RoboDK station: PenHolder.rdk

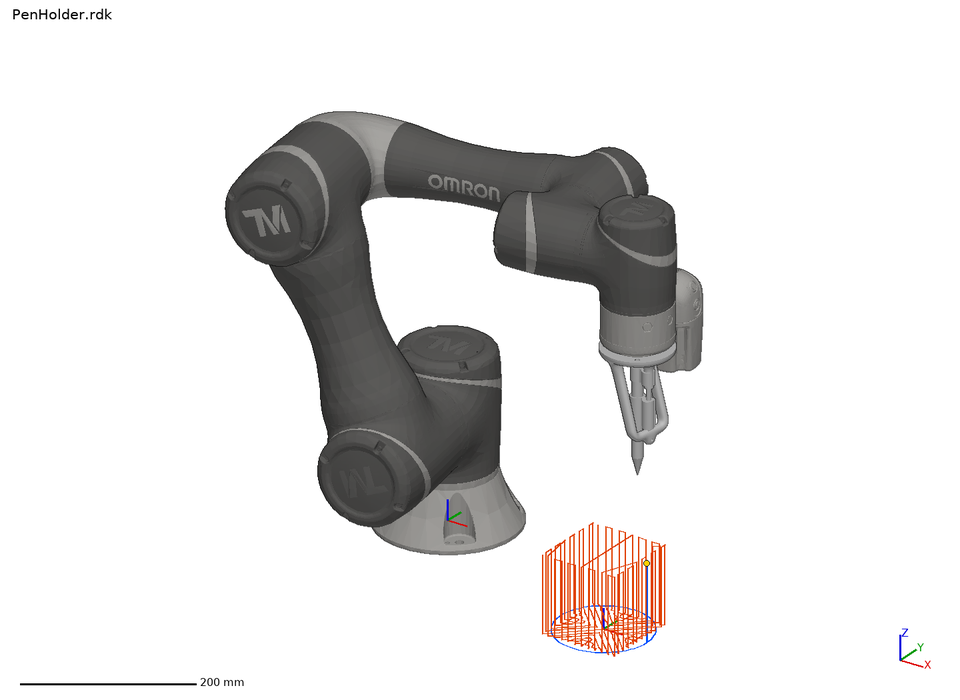
[picture v0: the station drawn from its stored meshes, robots at their saved joint values, targets as dots, program paths as lines]
Station PenHolder (saved by RoboDK 5.6.7). Poses are relative to the parent item; angles as X-Y-Z fixed-axis rotations.
  - frame Omron TM5-700 Base at (0, 0, 0) mm
    - robot Omron TM5-700: 6 axes, payload 6 kg, reach 700 mm, repeatability 0.05 mm, weight 22.1 kg
        modified DH rows (alpha deg, a mm, theta deg, d mm): 0, 0, 0, 145.2; 90, 0, 90, 0; 0, 329, 0, 0; 0, 311, -90, 122.3; -90, 0, 0, 106.5; 90, 0, 180, 114.15
        joint limits [-270, -180, -155, -180, -180, -270] to [270, 180, 155, 180, 180, 270]; home [0, 0, 90, -90, 90, 0]; saved at [8.928, -21.013, 110.905, 0.108, 90, -86.327]
      - tool PenHolderTCP, TCP at (0, 0, 163) mm, size 163 x 88.1 x 88.4 mm, geometry from PenHolderTCP.stl
  - frame Canvas at (306.28, -129, 0) mm
    - object circle at (0, 0, 0) mm, geometry from pter
    - object pattern at (0, 0, 0) mm, geometry from amag
  - machining project circle Settings: rotZ(0) | rotX(0)*rotY(0) | rotz(0) | onStart | onPathStart | onApproach | onPoint | onRetract | onFinish | SetRPM(%1) | SetTool(%1) | Extruder(%1) | default | default | OutOnMov(%1) | OutOffMov(%1) | onPathFinish | M_RunCode(%1)
  - program circle (86 instructions, listed below)
  - machining project pattern Settings: rotZ(0) | rotX(0)*rotY(0) | rotz(0) | onStart | onPathStart | onApproach | onPoint | onRetract | onFinish | SetRPM(%1) | SetTool(%1) | Extruder(%1) | default | default | OutOnMov(%1) | OutOffMov(%1) | onPathFinish | M_RunCode(%1)
  - program patternLinear (449 instructions, listed below)
  - Python program Prog3 (listed below)
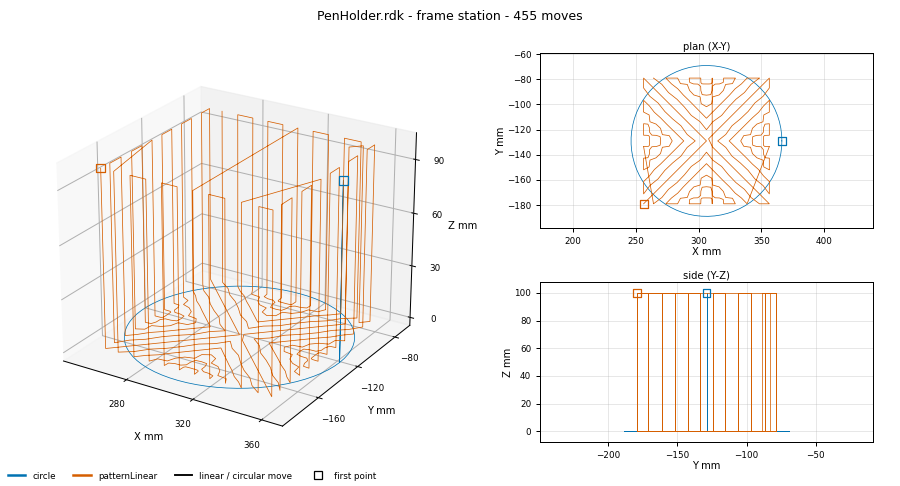
[picture p0: tool path of PenHolder.rdk in frame station, 455 of 455 moves have a stored position in this frame; points joined in program order, loops and branches not executed]

--- program circle (robot Omron TM5-700) ---
  Smooth(1)
  Set speed (1000.0 mm/s)
  Set Ref.: Canvas
  Set Tool: PenHolderTCP
  Show PenHolderTCP
  MoveJ 1 to (60, 0, 100) mm, rotated rx -180 ry 0 rz -180 deg; joints [-1.045, -5.926, 113.769, -17.843, 90, -91.045]
  MoveL 2 to (60, 0, 100) mm, rotated rx -180 ry 0 rz -180 deg; joints [-1.045, -5.926, 113.769, -17.843, 90, -91.045]
  MoveL 3 to (60, 0, 0) mm, rotated rx -180 ry 0 rz -180 deg; joints [-1.045, 3.646, 125.512, -39.158, 90, -91.045]
  MoveL 4 to (60, 0, 0) mm, rotated rx -180 ry 0 rz -180 deg; joints [-1.045, 3.646, 125.512, -39.158, 90, -91.045]
  Set speed (50.0 mm/s)
  MoveL 5 to (59.78, 5.16, 0) mm, rotated rx -180 ry 0 rz -180 deg; joints [-0.241, 3.314, 125.871, -39.185, 90, -90.241]
  MoveL 6 to (59.11, 10.28, 0) mm, rotated rx -180 ry 0 rz -180 deg; joints [0.562, 2.919, 126.295, -39.215, 90, -89.438]
  MoveL 7 to (58.01, 15.32, 0) mm, rotated rx -180 ry 0 rz -180 deg; joints [1.361, 2.462, 126.782, -39.244, 90, -88.639]
  MoveL 8 to (56.48, 20.25, 0) mm, rotated rx -180 ry 0 rz 180 deg; joints [2.153, 1.943, 127.328, -39.271, 90, -87.847]
  MoveL 9 to (54.53, 25.03, 0) mm, rotated rx -180 ry 0 rz -180 deg; joints [2.934, 1.364, 127.93, -39.294, 90, -87.066]
  MoveL 10 to (52.18, 29.63, 0) mm, rotated rx -180 ry 0 rz -180 deg; joints [3.7, 0.726, 128.584, -39.31, 90, -86.3]
  MoveL 11 to (49.44, 34, 0) mm, rotated rx -180 ry 0 rz -180 deg; joints [4.448, 0.029, 129.287, -39.316, 90, -85.552]
  MoveL 12 to (46.33, 38.13, 0) mm, rotated rx -180 ry 0 rz -180 deg; joints [5.173, -0.723, 130.033, -39.31, 90, -84.827]
  MoveL 13 to (42.88, 41.97, 0) mm, rotated rx -180 ry 0 rz -180 deg; joints [5.872, -1.529, 130.818, -39.288, 90, -84.128]
  MoveL 14 to (39.11, 45.5, 0) mm, rotated rx -180 ry 0 rz -180 deg; joints [6.54, -2.388, 131.636, -39.248, 90, -83.46]
  MoveL 15 to (35.06, 48.69, 0) mm, rotated rx -180 ry 0 rz -180 deg; joints [7.173, -3.295, 132.482, -39.187, 90, -82.827]
  MoveL 16 to (30.74, 51.53, 0) mm, rotated rx -180 ry 0 rz -180 deg; joints [7.765, -4.25, 133.351, -39.101, 90, -82.235]
  MoveL 17 to (26.2, 53.98, 0) mm, rotated rx -180 ry 0 rz -180 deg; joints [8.312, -5.247, 134.236, -38.989, 90, -81.688]
  MoveL 18 to (21.46, 56.03, 0) mm, rotated rx -180 ry 0 rz -180 deg; joints [8.809, -6.284, 135.131, -38.847, 90, -81.191]
  MoveL 19 to (16.57, 57.67, 0) mm, rotated rx -180 ry 0 rz -180 deg; joints [9.25, -7.355, 136.03, -38.675, 90, -80.75]
  MoveL 20 to (11.55, 58.88, 0) mm, rotated rx -180 ry 0 rz -180 deg; joints [9.63, -8.455, 136.925, -38.47, 90, -80.37]
  MoveL 21 to (6.44, 59.65, 0) mm, rotated rx -180 ry 0 rz -180 deg; joints [9.942, -9.577, 137.81, -38.233, 90, -80.058]
  MoveL 22 to (1.29, 59.99, 0) mm, rotated rx -180 ry 0 rz -180 deg; joints [10.182, -10.715, 138.678, -37.963, 90, -79.818]
  MoveL 23 to (-3.87, 59.88, 0) mm, rotated rx -180 ry 0 rz -180 deg; joints [10.343, -11.858, 139.522, -37.664, 90, -79.657]
  MoveL 24 to (-9, 59.32, 0) mm, rotated rx -180 ry 0 rz -180 deg; joints [10.42, -12.999, 140.335, -37.336, 90, -79.58]
  MoveL 25 to (-14.07, 58.33, 0) mm, rotated rx -180 ry 0 rz -180 deg; joints [10.408, -14.124, 141.11, -36.986, 90, -79.592]
  MoveL 26 to (-19.03, 56.9, 0) mm, rotated rx -180 ry 0 rz 180 deg; joints [10.3, -15.223, 141.841, -36.618, 90, -79.7]
  MoveL 27 to (-23.85, 55.06, 0) mm, rotated rx -180 ry 0 rz -180 deg; joints [10.094, -16.282, 142.522, -36.24, 90, -79.906]
  MoveL 28 to (-28.5, 52.8, 0) mm, rotated rx -180 ry 0 rz -180 deg; joints [9.785, -17.285, 143.146, -35.861, 90, -80.215]
  MoveL 29 to (-32.93, 50.16, 0) mm, rotated rx -180 ry 0 rz -180 deg; joints [9.371, -18.217, 143.709, -35.491, 90, -80.629]
  MoveL 30 to (-37.12, 47.14, 0) mm, rotated rx -180 ry 0 rz -180 deg; joints [8.851, -19.064, 144.204, -35.14, 90, -81.149]
  MoveL 31 to (-41.04, 43.77, 0) mm, rotated rx -180 ry 0 rz 180 deg; joints [8.226, -19.808, 144.629, -34.82, 90, -81.774]
  MoveL 32 to (-44.65, 40.08, 0) mm, rotated rx -180 ry 0 rz -180 deg; joints [7.498, -20.437, 144.979, -34.542, 90, -82.502]
  MoveL 33 to (-47.93, 36.1, 0) mm, rotated rx -180 ry 0 rz -180 deg; joints [6.674, -20.936, 145.252, -34.316, 90, -83.326]
  MoveL 34 to (-50.85, 31.84, 0) mm, rotated rx -180 ry 0 rz -180 deg; joints [5.76, -21.295, 145.446, -34.151, 90, -84.24]
  MoveL 35 to (-53.4, 27.35, 0) mm, rotated rx -180 ry 0 rz -180 deg; joints [4.765, -21.506, 145.558, -34.053, 90, -85.235]
  MoveL 36 to (-55.56, 22.66, 0) mm, rotated rx -180 ry 0 rz -180 deg; joints [3.701, -21.563, 145.588, -34.026, 90, -86.299]
  MoveL 37 to (-57.3, 17.8, 0) mm, rotated rx -180 ry 0 rz -180 deg; joints [2.582, -21.465, 145.537, -34.072, 90, -87.418]
  MoveL 38 to (-58.62, 12.81, 0) mm, rotated rx -180 ry 0 rz -180 deg; joints [1.422, -21.215, 145.403, -34.188, 90, -88.578]
  MoveL 39 to (-59.5, 7.72, 0) mm, rotated rx -180 ry 0 rz -180 deg; joints [0.238, -20.818, 145.188, -34.37, 90, -89.762]
  MoveL 40 to (-59.94, 2.58, 0) mm, rotated rx -180 ry 0 rz -180 deg; joints [-0.954, -20.284, 144.895, -34.611, 90, -90.954]
  MoveL 41 to (-59.94, -2.58, 0) mm, rotated rx -180 ry 0 rz -180 deg; joints [-2.138, -19.623, 144.524, -34.901, 90, -92.138]
  MoveL 42 to (-59.5, -7.72, 0) mm, rotated rx -180 ry 0 rz 180 deg; joints [-3.299, -18.85, 144.081, -35.23, 90, -93.299]
  MoveL 43 to (-58.62, -12.81, 0) mm, rotated rx -180 ry 0 rz -180 deg; joints [-4.421, -17.98, 143.567, -35.587, 90, -94.421]
  MoveL 44 to (-57.3, -17.8, 0) mm, rotated rx -180 ry 0 rz -180 deg; joints [-5.492, -17.027, 142.988, -35.961, 90, -95.492]
  MoveL 45 to (-55.56, -22.66, 0) mm, rotated rx -180 ry 0 rz -180 deg; joints [-6.501, -16.008, 142.348, -36.34, 90, -96.501]
  MoveL 46 to (-53.4, -27.35, 0) mm, rotated rx -180 ry 0 rz -180 deg; joints [-7.439, -14.938, 141.654, -36.716, 90, -97.439]
  MoveL 47 to (-50.85, -31.84, 0) mm, rotated rx -180 ry 0 rz -180 deg; joints [-8.297, -13.83, 140.911, -37.08, 90, -98.297]
  MoveL 48 to (-47.93, -36.1, 0) mm, rotated rx -180 ry 0 rz 180 deg; joints [-9.071, -12.7, 140.125, -37.425, 90, -99.071]
  MoveL 49 to (-44.65, -40.08, 0) mm, rotated rx -180 ry 0 rz 180 deg; joints [-9.757, -11.557, 139.303, -37.745, 90, -99.757]
  MoveL 50 to (-41.04, -43.77, 0) mm, rotated rx -180 ry 0 rz -180 deg; joints [-10.352, -10.414, 138.452, -38.037, 90, -100.352]
  MoveL 51 to (-37.12, -47.14, 0) mm, rotated rx -180 ry 0 rz -180 deg; joints [-10.855, -9.28, 137.579, -38.298, 90, -100.855]
  MoveL 52 to (-32.93, -50.16, 0) mm, rotated rx -180 ry 0 rz -180 deg; joints [-11.266, -8.163, 136.69, -38.527, 90, -101.266]
  MoveL 53 to (-28.5, -52.8, 0) mm, rotated rx -180 ry 0 rz -180 deg; joints [-11.587, -7.07, 135.793, -38.723, 90, -101.587]
  MoveL 54 to (-23.85, -55.06, 0) mm, rotated rx -180 ry 0 rz 180 deg; joints [-11.82, -6.008, 134.895, -38.887, 90, -101.82]
  MoveL 55 to (-19.03, -56.9, 0) mm, rotated rx -180 ry 0 rz -180 deg; joints [-11.967, -4.981, 134.002, -39.021, 90, -101.967]
  MoveL 56 to (-14.07, -58.33, 0) mm, rotated rx -180 ry 0 rz -180 deg; joints [-12.032, -3.995, 133.121, -39.126, 90, -102.032]
  MoveL 57 to (-9, -59.32, 0) mm, rotated rx -180 ry 0 rz 180 deg; joints [-12.017, -3.052, 132.257, -39.205, 90, -102.017]
  MoveL 58 to (-3.87, -59.88, 0) mm, rotated rx -180 ry 0 rz -180 deg; joints [-11.927, -2.157, 131.418, -39.261, 90, -101.927]
  MoveL 59 to (1.29, -59.99, 0) mm, rotated rx -180 ry 0 rz 180 deg; joints [-11.766, -1.312, 130.608, -39.296, 90, -101.766]
  MoveL 60 to (6.44, -59.65, 0) mm, rotated rx -180 ry 0 rz 180 deg; joints [-11.537, -0.52, 129.833, -39.313, 90, -101.537]
  MoveL 61 to (11.55, -58.88, 0) mm, rotated rx -180 ry 0 rz -180 deg; joints [-11.244, 0.218, 129.098, -39.316, 90, -101.244]
  MoveL 62 to (16.57, -57.67, 0) mm, rotated rx -180 ry 0 rz -180 deg; joints [-10.892, 0.899, 128.408, -39.307, 90, -100.892]
  MoveL 63 to (21.46, -56.03, 0) mm, rotated rx -180 ry 0 rz -180 deg; joints [-10.485, 1.522, 127.767, -39.289, 90, -100.485]
  MoveL 64 to (26.2, -53.98, 0) mm, rotated rx -180 ry 0 rz -180 deg; joints [-10.026, 2.085, 127.179, -39.264, 90, -100.026]
  MoveL 65 to (30.74, -51.53, 0) mm, rotated rx -180 ry 0 rz -180 deg; joints [-9.52, 2.588, 126.648, -39.236, 90, -99.52]
  MoveL 66 to (35.06, -48.69, 0) mm, rotated rx -180 ry 0 rz -180 deg; joints [-8.97, 3.029, 126.178, -39.207, 90, -98.97]
  MoveL 67 to (39.11, -45.5, 0) mm, rotated rx -180 ry 0 rz 180 deg; joints [-8.38, 3.407, 125.77, -39.178, 90, -98.38]
  MoveL 68 to (42.88, -41.97, 0) mm, rotated rx -180 ry 0 rz -180 deg; joints [-7.753, 3.722, 125.429, -39.151, 90, -97.753]
  MoveL 69 to (46.33, -38.13, 0) mm, rotated rx -180 ry 0 rz -180 deg; joints [-7.094, 3.973, 125.155, -39.128, 90, -97.094]
  MoveL 70 to (49.44, -34, 0) mm, rotated rx -180 ry 0 rz -180 deg; joints [-6.406, 4.16, 124.95, -39.11, 90, -96.406]
  MoveL 71 to (52.18, -29.63, 0) mm, rotated rx -180 ry 0 rz 180 deg; joints [-5.691, 4.282, 124.816, -39.098, 90, -95.691]
  MoveL 72 to (54.53, -25.03, 0) mm, rotated rx -180 ry 0 rz -180 deg; joints [-4.954, 4.338, 124.754, -39.092, 90, -94.954]
  MoveL 73 to (56.48, -20.25, 0) mm, rotated rx -180 ry 0 rz -180 deg; joints [-4.197, 4.33, 124.764, -39.093, 90, -94.197]
  MoveL 74 to (58.01, -15.32, 0) mm, rotated rx -180 ry 0 rz 180 deg; joints [-3.425, 4.256, 124.845, -39.101, 90, -93.425]
  MoveL 75 to (59.11, -10.28, 0) mm, rotated rx -180 ry 0 rz -180 deg; joints [-2.64, 4.117, 124.997, -39.114, 90, -92.64]
  MoveL 76 to (59.78, -5.16, 0) mm, rotated rx -180 ry 0 rz -180 deg; joints [-1.846, 3.914, 125.22, -39.134, 90, -91.846]
  MoveL 77 to (60, 0, 0) mm, rotated rx -180 ry 0 rz -180 deg; joints [-1.045, 3.646, 125.512, -39.158, 90, -91.045]
  Set speed (1000.0 mm/s)
  MoveL 78 to (60, 0, 0) mm, rotated rx -180 ry 0 rz -180 deg; joints [-1.045, 3.646, 125.512, -39.158, 90, -91.045]
  MoveL 79 to (60, 0, 100) mm, rotated rx -180 ry 0 rz -180 deg; joints [-1.045, -5.926, 113.769, -17.843, 90, -91.045]

--- program patternLinear (robot Omron TM5-700) ---
  Smooth(1)
  Set speed (1000.0 mm/s)
  Set Ref.: Canvas
  Set Tool: PenHolderTCP
  Show PenHolderTCP
  MoveJ 1 to (-50, -50, 100) mm, rotated rx -180 ry 0 rz -180 deg; joints [-11.902, -21.555, 125.328, -13.773, 90, -101.902]
  MoveL 2 to (-50, -50, 100) mm, rotated rx -180 ry 0 rz -180 deg; joints [-11.902, -21.555, 125.328, -13.773, 90, -101.902]
  MoveL 3 to (-50, -50, 0) mm, rotated rx -180 ry 0 rz -180 deg; joints [-11.902, -11.308, 139.12, -37.811, 90, -101.902]
  MoveL 4 to (-50, -50, 0) mm, rotated rx -180 ry 0 rz -180 deg; joints [-11.902, -11.308, 139.12, -37.811, 90, -101.902]
  Set speed (50.0 mm/s)
  MoveL 5 to (-7.14, -7.14, 0) mm, rotated rx -180 ry 0 rz -180 deg; joints [-2.625, -7.772, 136.372, -38.6, 90, -92.625]
  MoveL 6 to (0, 0, 0) mm, rotated rx -180 ry 0 rz -180 deg; joints [-1.248, -6.997, 135.732, -38.735, 90, -91.248]
  MoveL 7 to (-50, 50, 0) mm, rotated rx -180 ry 0 rz -180 deg; joints [9.999, -22.769, 146.216, -33.447, 90, -80.001]
  Set speed (1000.0 mm/s)
  MoveL 8 to (-50, 50, 0) mm, rotated rx -180 ry 0 rz -180 deg; joints [9.999, -22.769, 146.216, -33.447, 90, -80.001]
  MoveL 9 to (-50, 50, 100) mm, rotated rx -180 ry 0 rz -180 deg; joints [9.999, -32.206, 130.792, -8.586, 90, -80.001]
  Set speed (1000.0 mm/s)
  MoveL 10 to (-50, 42.13, 100) mm, rotated rx -180 ry 0 rz 180 deg; joints [8.143, -31.588, 130.523, -8.935, 90, -81.857]
  MoveL 11 to (-50, 42.13, 0) mm, rotated rx -180 ry 0 rz 180 deg; joints [8.143, -22.062, 145.851, -33.789, 90, -81.857]
  MoveL 12 to (-50, 42.13, 0) mm, rotated rx -180 ry 0 rz 180 deg; joints [8.143, -22.062, 145.851, -33.789, 90, -81.857]
  Set speed (50.0 mm/s)
  MoveL 13 to (-45.03, 35.49, 0) mm, rotated rx -180 ry 0 rz -180 deg; joints [6.459, -20.118, 144.802, -34.684, 90, -83.541]
  MoveL 14 to (-38.5, 30.21, 0) mm, rotated rx -180 ry 0 rz 180 deg; joints [5.121, -17.972, 143.562, -35.59, 90, -84.879]
  MoveL 15 to (-33.12, 23.42, 0) mm, rotated rx -180 ry 0 rz -180 deg; joints [3.551, -16.051, 142.375, -36.325, 90, -86.449]
  MoveL 16 to (-26.96, 17.54, 0) mm, rotated rx -180 ry 0 rz -180 deg; joints [2.241, -14.099, 141.093, -36.994, 90, -87.759]
  MoveL 17 to (-20.31, 12.08, 0) mm, rotated rx -180 ry 0 rz -180 deg; joints [1.081, -12.149, 139.732, -37.583, 90, -88.919]
  MoveL 18 to (-15.34, 5.14, 0) mm, rotated rx -180 ry 0 rz -180 deg; joints [-0.307, -10.493, 138.511, -38.018, 90, -90.307]
  MoveL 19 to (-8.95, 0, 0) mm, rotated rx -180 ry 0 rz -180 deg; joints [-1.285, -8.749, 137.159, -38.411, 90, -91.285]
  MoveL 20 to (-15.34, -5.14, 0) mm, rotated rx -180 ry 0 rz 180 deg; joints [-2.311, -9.566, 137.801, -38.235, 90, -92.311]
  MoveL 21 to (-20.31, -12.08, 0) mm, rotated rx -180 ry 0 rz -180 deg; joints [-3.706, -9.896, 138.056, -38.16, 90, -93.706]
  MoveL 22 to (-26.96, -17.54, 0) mm, rotated rx -180 ry 0 rz 180 deg; joints [-4.869, -10.668, 138.643, -37.975, 90, -94.869]
  MoveL 23 to (-33.12, -23.42, 0) mm, rotated rx -180 ry 0 rz -180 deg; joints [-6.145, -11.262, 139.085, -37.824, 90, -96.145]
  MoveL 24 to (-38.5, -30.21, 0) mm, rotated rx -180 ry 0 rz -180 deg; joints [-7.619, -11.553, 139.3, -37.746, 90, -97.619]
  MoveL 25 to (-45.03, -35.49, 0) mm, rotated rx -180 ry 0 rz -180 deg; joints [-8.859, -12.203, 139.771, -37.568, 90, -98.859]
  MoveL 26 to (-50, -42.13, 0) mm, rotated rx -180 ry 0 rz 180 deg; joints [-10.35, -12.334, 139.864, -37.531, 90, -100.35]
  Set speed (1000.0 mm/s)
  MoveL 27 to (-50, -42.13, 0) mm, rotated rx -180 ry 0 rz 180 deg; joints [-10.35, -12.334, 139.864, -37.531, 90, -100.35]
  MoveL 28 to (-50, -42.13, 100) mm, rotated rx -180 ry 0 rz 180 deg; joints [-10.35, -22.561, 125.923, -13.362, 90, -100.35]
  Set speed (1000.0 mm/s)
  MoveL 29 to (-50, -32.32, 100) mm, rotated rx -180 ry 0 rz -180 deg; joints [-8.369, -23.786, 126.624, -12.838, 90, -98.369]
  MoveL 30 to (-50, -32.32, 0) mm, rotated rx -180 ry 0 rz -180 deg; joints [-8.369, -13.596, 140.75, -37.154, 90, -98.369]
  MoveL 31 to (-50, -32.32, 0) mm, rotated rx -180 ry 0 rz -180 deg; joints [-8.369, -13.596, 140.75, -37.154, 90, -98.369]
  Set speed (50.0 mm/s)
  MoveL 32 to (-45.4, -27.84, 0) mm, rotated rx -180 ry 0 rz -180 deg; joints [-7.325, -13.221, 140.49, -37.269, 90, -97.325]
  MoveL 33 to (-41.5, -22.82, 0) mm, rotated rx -180 ry 0 rz -180 deg; joints [-6.208, -13.025, 140.354, -37.328, 90, -96.208]
  MoveL 34 to (-36.52, -18.38, 0) mm, rotated rx -180 ry 0 rz -180 deg; joints [-5.205, -12.513, 139.992, -37.479, 90, -95.205]
  MoveL 35 to (-22.58, -4.47, 0) mm, rotated rx -180 ry 0 rz -180 deg; joints [-2.237, -11.097, 138.963, -37.866, 90, -92.237]
  MoveL 36 to (-18.05, 0, 0) mm, rotated rx -180 ry 0 rz -180 deg; joints [-1.325, -10.589, 138.583, -37.995, 90, -91.325]
  MoveL 37 to (-31.87, 13.57, 0) mm, rotated rx -180 ry 0 rz -180 deg; joints [1.442, -14.841, 141.59, -36.749, 90, -88.558]
  MoveL 38 to (-36.52, 18.38, 0) mm, rotated rx -180 ry 0 rz 180 deg; joints [2.504, -16.38, 142.584, -36.204, 90, -87.496]
  MoveL 39 to (-41.5, 22.82, 0) mm, rotated rx -180 ry 0 rz -180 deg; joints [3.534, -18.009, 143.585, -35.575, 90, -86.466]
  MoveL 40 to (-45.4, 27.84, 0) mm, rotated rx -180 ry 0 rz -180 deg; joints [4.724, -19.478, 144.442, -34.964, 90, -85.276]
  MoveL 41 to (-50, 32.32, 0) mm, rotated rx -180 ry 0 rz -180 deg; joints [5.85, -21.117, 145.35, -34.233, 90, -84.15]
  Set speed (1000.0 mm/s)
  MoveL 42 to (-50, 32.32, 0) mm, rotated rx -180 ry 0 rz -180 deg; joints [5.85, -21.117, 145.35, -34.233, 90, -84.15]
  MoveL 43 to (-50, 32.32, 100) mm, rotated rx -180 ry 0 rz -180 deg; joints [5.85, -30.754, 130.152, -9.398, 90, -84.15]
  Set speed (1000.0 mm/s)
  MoveL 44 to (-50, 22.96, 100) mm, rotated rx -180 ry 0 rz -180 deg; joints [3.687, -29.894, 129.758, -9.864, 90, -86.313]
  MoveL 45 to (-50, 22.96, 0) mm, rotated rx -180 ry 0 rz -180 deg; joints [3.687, -20.153, 144.822, -34.669, 90, -86.313]
  MoveL 46 to (-50, 22.96, 0) mm, rotated rx -180 ry 0 rz -180 deg; joints [3.687, -20.153, 144.822, -34.669, 90, -86.313]
  Set speed (50.0 mm/s)
  MoveL 47 to (-45.6, 20.68, 0) mm, rotated rx -180 ry 0 rz -180 deg; joints [3.11, -18.807, 144.055, -35.248, 90, -86.89]
  MoveL 48 to (-44.95, 15.25, 0) mm, rotated rx -180 ry 0 rz -180 deg; joints [1.888, -18.079, 143.626, -35.547, 90, -88.112]
  MoveL 49 to (-40.17, 13.45, 0) mm, rotated rx -180 ry 0 rz -180 deg; joints [1.46, -16.749, 142.815, -36.066, 90, -88.54]
  MoveL 50 to (-36.57, 10.06, 0) mm, rotated rx -180 ry 0 rz -180 deg; joints [0.716, -15.57, 142.067, -36.497, 90, -89.284]
  MoveL 51 to (-35.06, 5.02, 0) mm, rotated rx -180 ry 0 rz -180 deg; joints [-0.354, -14.717, 141.508, -36.791, 90, -90.354]
  MoveL 52 to (-29.65, 4.22, 0) mm, rotated rx -180 ry 0 rz -180 deg; joints [-0.513, -13.442, 140.644, -37.202, 90, -90.513]
  MoveL 53 to (-27.24, 0, 0) mm, rotated rx -180 ry 0 rz -180 deg; joints [-1.368, -12.507, 139.988, -37.481, 90, -91.368]
  MoveL 54 to (-29.65, -4.22, 0) mm, rotated rx -180 ry 0 rz 180 deg; joints [-2.242, -12.597, 140.052, -37.455, 90, -92.242]
  MoveL 55 to (-35.06, -5.02, 0) mm, rotated rx -180 ry 0 rz -180 deg; joints [-2.452, -13.668, 140.799, -37.131, 90, -92.452]
  MoveL 56 to (-36.57, -10.06, 0) mm, rotated rx -180 ry 0 rz -180 deg; joints [-3.508, -13.447, 140.647, -37.2, 90, -93.508]
  MoveL 57 to (-40.17, -13.45, 0) mm, rotated rx -180 ry 0 rz -180 deg; joints [-4.257, -13.833, 140.913, -37.079, 90, -94.257]
  MoveL 58 to (-44.95, -15.25, 0) mm, rotated rx -180 ry 0 rz -180 deg; joints [-4.71, -14.645, 141.46, -36.815, 90, -94.71]
  MoveL 59 to (-45.6, -20.68, 0) mm, rotated rx -180 ry 0 rz -180 deg; joints [-5.858, -14.134, 141.117, -36.983, 90, -95.858]
  MoveL 60 to (-50, -22.96, 0) mm, rotated rx -180 ry 0 rz -180 deg; joints [-6.431, -14.781, 141.55, -36.769, 90, -96.431]
  Set speed (1000.0 mm/s)
  MoveL 61 to (-50, -22.96, 0) mm, rotated rx -180 ry 0 rz -180 deg; joints [-6.431, -14.781, 141.55, -36.769, 90, -96.431]
  MoveL 62 to (-50, -22.96, 100) mm, rotated rx -180 ry 0 rz -180 deg; joints [-6.431, -24.922, 127.253, -12.33, 90, -96.431]
  Set speed (1000.0 mm/s)
  MoveL 63 to (-50, -13.71, 100) mm, rotated rx -180 ry 0 rz -180 deg; joints [-4.47, -26.01, 127.835, -11.824, 90, -94.47]
  MoveL 64 to (-50, -13.71, 0) mm, rotated rx -180 ry 0 rz -180 deg; joints [-4.47, -15.93, 142.299, -36.368, 90, -94.47]
  MoveL 65 to (-50, -13.71, 0) mm, rotated rx -180 ry 0 rz -180 deg; joints [-4.47, -15.93, 142.299, -36.368, 90, -94.47]
  Set speed (50.0 mm/s)
  MoveL 66 to (-46.56, -13.35, 0) mm, rotated rx -180 ry 0 rz -180 deg; joints [-4.337, -15.221, 141.84, -36.619, 90, -94.337]
  MoveL 67 to (-45.35, -10.35, 0) mm, rotated rx -180 ry 0 rz -180 deg; joints [-3.684, -15.311, 141.899, -36.588, 90, -93.684]
  MoveL 68 to (-45.22, -6.89, 0) mm, rotated rx -180 ry 0 rz -180 deg; joints [-2.945, -15.685, 142.141, -36.456, 90, -92.945]
  MoveL 69 to (-43.44, -4.62, 0) mm, rotated rx -180 ry 0 rz -180 deg; joints [-2.442, -15.549, 142.053, -36.505, 90, -92.442]
  MoveL 70 to (-39.98, -4.45, 0) mm, rotated rx -180 ry 0 rz -180 deg; joints [-2.375, -14.801, 141.563, -36.763, 90, -92.375]
  MoveL 71 to (-36.83, -3.42, 0) mm, rotated rx -180 ry 0 rz -180 deg; joints [-2.133, -14.223, 141.177, -36.954, 90, -92.133]
  MoveL 72 to (-36.42, 0, 0) mm, rotated rx -180 ry 0 rz -180 deg; joints [-1.415, -14.497, 141.361, -36.864, 90, -91.415]
  MoveL 73 to (-36.83, 3.42, 0) mm, rotated rx -180 ry 0 rz -180 deg; joints [-0.696, -14.946, 141.66, -36.713, 90, -90.696]
  MoveL 74 to (-39.98, 4.45, 0) mm, rotated rx -180 ry 0 rz 180 deg; joints [-0.484, -15.765, 142.193, -36.428, 90, -90.484]
  MoveL 75 to (-43.44, 4.62, 0) mm, rotated rx -180 ry 0 rz -180 deg; joints [-0.453, -16.578, 142.709, -36.13, 90, -90.453]
  MoveL 76 to (-45.22, 6.89, 0) mm, rotated rx -180 ry 0 rz -180 deg; joints [0.042, -17.243, 143.121, -35.878, 90, -89.958]
  MoveL 77 to (-45.35, 10.35, 0) mm, rotated rx -180 ry 0 rz -180 deg; joints [0.805, -17.653, 143.37, -35.717, 90, -89.195]
  MoveL 78 to (-46.56, 13.35, 0) mm, rotated rx -180 ry 0 rz -180 deg; joints [1.474, -18.267, 143.738, -35.471, 90, -88.526]
  MoveL 79 to (-50, 13.71, 0) mm, rotated rx -180 ry 0 rz 180 deg; joints [1.576, -19.149, 144.253, -35.105, 90, -88.424]
  Set speed (1000.0 mm/s)
  MoveL 80 to (-50, 13.71, 0) mm, rotated rx -180 ry 0 rz 180 deg; joints [1.576, -19.149, 144.253, -35.105, 90, -88.424]
  MoveL 81 to (-50, 13.71, 100) mm, rotated rx -180 ry 0 rz 180 deg; joints [1.576, -28.986, 129.329, -10.343, 90, -88.424]
  Set speed (1000.0 mm/s)
  MoveL 82 to (-50, 4.55, 100) mm, rotated rx -180 ry 0 rz -180 deg; joints [-0.48, -28.037, 128.868, -10.831, 90, -90.48]
  MoveL 83 to (-50, 4.55, 0) mm, rotated rx -180 ry 0 rz -180 deg; joints [-0.48, -18.11, 143.645, -35.535, 90, -90.48]
  MoveL 84 to (-50, 4.55, 0) mm, rotated rx -180 ry 0 rz -180 deg; joints [-0.48, -18.11, 143.645, -35.535, 90, -90.48]
  Set speed (50.0 mm/s)
  MoveL 85 to (-48.78, 4.53, 0) mm, rotated rx -180 ry 0 rz -180 deg; joints [-0.482, -17.816, 143.469, -35.652, 90, -90.482]
  MoveL 86 to (-47.55, 4.49, 0) mm, rotated rx -180 ry 0 rz -180 deg; joints [-0.488, -17.523, 143.292, -35.768, 90, -90.488]
  MoveL 87 to (-46.33, 4.39, 0) mm, rotated rx -180 ry 0 rz -180 deg; joints [-0.508, -17.225, 143.11, -35.885, 90, -90.508]
  MoveL 88 to (-45.46, 3.67, 0) mm, rotated rx -180 ry 0 rz -180 deg; joints [-0.665, -16.942, 142.935, -35.993, 90, -90.665]
  MoveL 89 to (-45.34, 2.45, 0) mm, rotated rx -180 ry 0 rz -180 deg; joints [-0.93, -16.777, 142.833, -36.056, 90, -90.93]
  MoveL 90 to (-45.3, -1.23, 0) mm, rotated rx -180 ry 0 rz 180 deg; joints [-1.727, -16.354, 142.568, -36.214, 90, -91.727]
  MoveL 91 to (-45.34, -2.45, 0) mm, rotated rx -180 ry 0 rz -180 deg; joints [-1.992, -16.222, 142.484, -36.262, 90, -91.992]
  MoveL 92 to (-45.46, -3.67, 0) mm, rotated rx -180 ry 0 rz -180 deg; joints [-2.256, -16.111, 142.414, -36.303, 90, -92.256]
  MoveL 93 to (-46.33, -4.39, 0) mm, rotated rx -180 ry 0 rz -180 deg; joints [-2.419, -16.223, 142.485, -36.262, 90, -92.419]
  MoveL 94 to (-47.55, -4.49, 0) mm, rotated rx -180 ry 0 rz -180 deg; joints [-2.452, -16.488, 142.652, -36.164, 90, -92.452]
  MoveL 95 to (-50, -4.55, 0) mm, rotated rx -180 ry 0 rz -180 deg; joints [-2.488, -17.04, 142.996, -35.956, 90, -92.488]
  Set speed (1000.0 mm/s)
  MoveL 96 to (-50, -4.55, 0) mm, rotated rx -180 ry 0 rz -180 deg; joints [-2.488, -17.04, 142.996, -35.956, 90, -92.488]
  MoveL 97 to (-50, -4.55, 100) mm, rotated rx -180 ry 0 rz -180 deg; joints [-2.488, -27.048, 128.372, -11.324, 90, -92.488]
  Set speed (1000.0 mm/s)
  MoveL 98 to (-42.13, -50, 100) mm, rotated rx -180 ry 0 rz -180 deg; joints [-11.586, -20.105, 124.44, -14.335, 90, -101.586]
  MoveL 99 to (-42.13, -50, 0) mm, rotated rx -180 ry 0 rz 180 deg; joints [-11.586, -9.849, 138.02, -38.171, 90, -101.586]
  MoveL 100 to (-42.13, -50, 0) mm, rotated rx -180 ry 0 rz 180 deg; joints [-11.586, -9.849, 138.02, -38.171, 90, -101.586]
  Set speed (50.0 mm/s)
  MoveL 101 to (-35.49, -45.03, 0) mm, rotated rx -180 ry 0 rz -180 deg; joints [-10.398, -9.233, 137.541, -38.309, 90, -100.398]
  MoveL 102 to (-30.21, -38.5, 0) mm, rotated rx -180 ry 0 rz -180 deg; joints [-8.991, -9.009, 137.365, -38.356, 90, -98.991]
  MoveL 103 to (-23.42, -33.12, 0) mm, rotated rx -180 ry 0 rz -180 deg; joints [-7.787, -8.335, 136.829, -38.494, 90, -97.787]
  MoveL 104 to (-17.54, -26.96, 0) mm, rotated rx -180 ry 0 rz -180 deg; joints [-6.495, -7.877, 136.458, -38.581, 90, -96.495]
  MoveL 105 to (-12.08, -20.31, 0) mm, rotated rx -180 ry 0 rz -180 deg; joints [-5.149, -7.505, 136.153, -38.648, 90, -95.149]
  MoveL 106 to (-5.14, -15.34, 0) mm, rotated rx -180 ry 0 rz -180 deg; joints [-4.127, -6.661, 135.45, -38.789, 90, -94.127]
  MoveL 107 to (0, -8.95, 0) mm, rotated rx -180 ry 0 rz 180 deg; joints [-2.896, -6.254, 135.106, -38.852, 90, -92.896]
  MoveL 108 to (5.14, -15.34, 0) mm, rotated rx -180 ry 0 rz -180 deg; joints [-3.995, -4.762, 133.809, -39.046, 90, -93.995]
  MoveL 109 to (12.08, -20.31, 0) mm, rotated rx -180 ry 0 rz -180 deg; joints [-4.773, -3.106, 132.307, -39.201, 90, -94.773]
  MoveL 110 to (17.54, -26.96, 0) mm, rotated rx -180 ry 0 rz -180 deg; joints [-5.823, -1.61, 130.895, -39.285, 90, -95.823]
  MoveL 111 to (23.42, -33.12, 0) mm, rotated rx -180 ry 0 rz -180 deg; joints [-6.741, -0.115, 129.431, -39.316, 90, -96.741]
  MoveL 112 to (30.21, -38.5, 0) mm, rotated rx -180 ry 0 rz 180 deg; joints [-7.476, 1.433, 127.858, -39.292, 90, -97.476]
  MoveL 113 to (35.49, -45.03, 0) mm, rotated rx -180 ry 0 rz -180 deg; joints [-8.39, 2.802, 126.421, -39.223, 90, -98.39]
  MoveL 114 to (42.13, -50, 0) mm, rotated rx -180 ry 0 rz -180 deg; joints [-8.999, 4.232, 124.871, -39.103, 90, -98.999]
  Set speed (1000.0 mm/s)
  MoveL 115 to (42.13, -50, 0) mm, rotated rx -180 ry 0 rz -180 deg; joints [-8.999, 4.232, 124.871, -39.103, 90, -98.999]
  MoveL 116 to (42.13, -50, 100) mm, rotated rx -180 ry 0 rz -180 deg; joints [-8.999, -5.286, 113.198, -17.912, 90, -98.999]
  Set speed (1000.0 mm/s)
  MoveL 117 to (50, -50, 100) mm, rotated rx -180 ry 0 rz -180 deg; joints [-8.813, -3.961, 111.992, -18.031, 90, -98.813]
  MoveL 118 to (50, -50, 0) mm, rotated rx -180 ry 0 rz -180 deg; joints [-8.813, 5.439, 123.525, -38.964, 90, -98.813]
  MoveL 119 to (50, -50, 0) mm, rotated rx -180 ry 0 rz -180 deg; joints [-8.813, 5.439, 123.525, -38.964, 90, -98.813]
  Set speed (50.0 mm/s)
  MoveL 120 to (4.79, -4.79, 0) mm, rotated rx -180 ry 0 rz 180 deg; joints [-2.101, -5.698, 134.628, -38.93, 90, -92.101]
  MoveL 121 to (1.67, 1.67, 0) mm, rotated rx -180 ry 0 rz -180 deg; joints [-0.934, -6.809, 135.575, -38.766, 90, -90.934]
  MoveL 122 to (8.12, 8.12, 0) mm, rotated rx -180 ry 0 rz -180 deg; joints [0.26, -6.063, 134.942, -38.879, 90, -89.74]
  MoveL 123 to (40.42, 40.42, 0) mm, rotated rx -180 ry 0 rz -180 deg; joints [5.652, -1.911, 131.184, -39.273, 90, -84.348]
  Set speed (1000.0 mm/s)
  MoveL 124 to (40.42, 40.42, 0) mm, rotated rx -180 ry 0 rz -180 deg; joints [5.652, -1.911, 131.184, -39.273, 90, -84.348]
  MoveL 125 to (40.42, 40.42, 100) mm, rotated rx -180 ry 0 rz -180 deg; joints [5.652, -11.913, 118.728, -16.814, 90, -84.348]
  Set speed (1000.0 mm/s)
  MoveL 126 to (45.76, 45.76, 100) mm, rotated rx -180 ry 0 rz -180 deg; joints [6.456, -11.126, 118.114, -16.988, 90, -83.544]
  MoveL 127 to (45.76, 45.76, 0) mm, rotated rx -180 ry 0 rz -180 deg; joints [6.456, -1.17, 130.47, -39.3, 90, -83.544]
  MoveL 128 to (45.76, 45.76, 0) mm, rotated rx -180 ry 0 rz -180 deg; joints [6.456, -1.17, 130.47, -39.3, 90, -83.544]
  Set speed (50.0 mm/s)
  MoveL 129 to (50, 50, 0) mm, rotated rx -180 ry 0 rz -180 deg; joints [7.078, -0.573, 129.885, -39.312, 90, -82.922]
  Set speed (1000.0 mm/s)
  MoveL 130 to (50, 50, 0) mm, rotated rx -180 ry 0 rz -180 deg; joints [7.078, -0.573, 129.885, -39.312, 90, -82.922]
  MoveL 131 to (50, 50, 100) mm, rotated rx -180 ry 0 rz -180 deg; joints [7.078, -10.488, 117.609, -17.121, 90, -82.922]
  Set speed (1000.0 mm/s)
  MoveL 132 to (50, 42.13, 100) mm, rotated rx -180 ry 0 rz -180 deg; joints [5.778, -10.133, 117.324, -17.191, 90, -84.222]
  MoveL 133 to (50, 42.13, 0) mm, rotated rx -180 ry 0 rz -180 deg; joints [5.778, -0.241, 129.557, -39.316, 90, -84.222]
  MoveL 134 to (50, 42.13, 0) mm, rotated rx -180 ry 0 rz -180 deg; joints [5.778, -0.241, 129.557, -39.316, 90, -84.222]
  Set speed (50.0 mm/s)
  MoveL 135 to (45.03, 35.49, 0) mm, rotated rx -180 ry 0 rz -180 deg; joints [4.754, -0.833, 130.141, -39.308, 90, -85.246]
  MoveL 136 to (38.5, 30.21, 0) mm, rotated rx -180 ry 0 rz -180 deg; joints [3.949, -1.755, 131.034, -39.28, 90, -86.051]
  MoveL 137 to (33.12, 23.42, 0) mm, rotated rx -180 ry 0 rz -180 deg; joints [2.845, -2.369, 131.618, -39.249, 90, -87.155]
  MoveL 138 to (26.96, 17.54, 0) mm, rotated rx -180 ry 0 rz -180 deg; joints [1.874, -3.153, 132.351, -39.198, 90, -88.126]
  MoveL 139 to (20.31, 12.08, 0) mm, rotated rx -180 ry 0 rz -180 deg; joints [0.946, -4.037, 133.159, -39.122, 90, -89.054]
  MoveL 140 to (15.34, 5.14, 0) mm, rotated rx -180 ry 0 rz 180 deg; joints [-0.278, -4.481, 133.559, -39.077, 90, -90.278]
  MoveL 141 to (8.95, 0, 0) mm, rotated rx -180 ry 0 rz -180 deg; joints [-1.213, -5.295, 134.278, -38.983, 90, -91.213]
  MoveL 142 to (15.34, -5.14, 0) mm, rotated rx -180 ry 0 rz -180 deg; joints [-2.094, -3.723, 132.874, -39.151, 90, -92.094]
  MoveL 143 to (20.31, -12.08, 0) mm, rotated rx -180 ry 0 rz -180 deg; joints [-3.256, -2.309, 131.562, -39.253, 90, -93.256]
  MoveL 144 to (26.96, -17.54, 0) mm, rotated rx -180 ry 0 rz -180 deg; joints [-4.106, -0.741, 130.05, -39.31, 90, -94.106]
  MoveL 145 to (33.12, -23.42, 0) mm, rotated rx -180 ry 0 rz -180 deg; joints [-4.993, 0.739, 128.57, -39.31, 90, -94.993]
  MoveL 146 to (38.5, -30.21, 0) mm, rotated rx -180 ry 0 rz -180 deg; joints [-6, 2.132, 127.13, -39.262, 90, -96]
  MoveL 147 to (45.03, -35.49, 0) mm, rotated rx -180 ry 0 rz -180 deg; joints [-6.713, 3.573, 125.592, -39.164, 90, -96.713]
  MoveL 148 to (50, -42.13, 0) mm, rotated rx -180 ry 0 rz -180 deg; joints [-7.631, 4.844, 124.193, -39.037, 90, -97.631]
  Set speed (1000.0 mm/s)
  MoveL 149 to (50, -42.13, 0) mm, rotated rx -180 ry 0 rz -180 deg; joints [-7.631, 4.844, 124.193, -39.037, 90, -97.631]
  MoveL 150 to (50, -42.13, 100) mm, rotated rx -180 ry 0 rz -180 deg; joints [-7.631, -4.614, 112.591, -17.977, 90, -97.631]
  Set speed (1000.0 mm/s)
  MoveL 151 to (50, -32.32, 100) mm, rotated rx -180 ry 0 rz -180 deg; joints [-6.138, -5.399, 113.3, -17.9, 90, -96.138]
  MoveL 152 to (50, -32.32, 0) mm, rotated rx -180 ry 0 rz -180 deg; joints [-6.138, 4.128, 124.985, -39.113, 90, -96.138]
  MoveL 153 to (50, -32.32, 0) mm, rotated rx -180 ry 0 rz -180 deg; joints [-6.138, 4.128, 124.985, -39.113, 90, -96.138]
  Set speed (50.0 mm/s)
  MoveL 154 to (45.4, -27.84, 0) mm, rotated rx -180 ry 0 rz -180 deg; joints [-5.518, 3.073, 126.131, -39.204, 90, -95.518]
  MoveL 155 to (41.5, -22.82, 0) mm, rotated rx -180 ry 0 rz -180 deg; joints [-4.782, 2.08, 127.185, -39.265, 90, -94.782]
  MoveL 156 to (36.52, -18.38, 0) mm, rotated rx -180 ry 0 rz -180 deg; joints [-4.132, 0.938, 128.368, -39.306, 90, -94.132]
  MoveL 157 to (31.87, -13.57, 0) mm, rotated rx -180 ry 0 rz 180 deg; joints [-3.395, -0.194, 129.51, -39.316, 90, -93.395]
  MoveL 158 to (18.05, 0, 0) mm, rotated rx -180 ry 0 rz -180 deg; joints [-1.179, -3.611, 132.772, -39.161, 90, -91.179]
  MoveL 159 to (22.58, 4.47, 0) mm, rotated rx -180 ry 0 rz -180 deg; joints [-0.387, -3.103, 132.304, -39.202, 90, -90.387]
  MoveL 160 to (36.52, 18.38, 0) mm, rotated rx -180 ry 0 rz -180 deg; joints [1.963, -1.461, 130.751, -39.291, 90, -88.037]
  MoveL 161 to (41.5, 22.82, 0) mm, rotated rx -180 ry 0 rz -180 deg; joints [2.676, -0.818, 130.126, -39.308, 90, -87.324]
  MoveL 162 to (45.4, 27.84, 0) mm, rotated rx -180 ry 0 rz -180 deg; joints [3.477, -0.386, 129.7, -39.315, 90, -86.523]
  MoveL 163 to (50, 32.32, 0) mm, rotated rx -180 ry 0 rz -180 deg; joints [4.164, 0.211, 129.105, -39.316, 90, -85.836]
  Set speed (1000.0 mm/s)
  MoveL 164 to (50, 32.32, 0) mm, rotated rx -180 ry 0 rz -180 deg; joints [4.164, 0.211, 129.105, -39.316, 90, -85.836]
  MoveL 165 to (50, 32.32, 100) mm, rotated rx -180 ry 0 rz -180 deg; joints [4.164, -9.648, 116.931, -17.283, 90, -85.836]
  Set speed (1000.0 mm/s)
  MoveL 166 to (50, 22.96, 100) mm, rotated rx -180 ry 0 rz -180 deg; joints [2.634, -9.143, 116.518, -17.375, 90, -87.366]
  MoveL 167 to (50, 22.96, 0) mm, rotated rx -180 ry 0 rz -180 deg; joints [2.634, 0.68, 128.631, -39.311, 90, -87.366]
  MoveL 168 to (50, 22.96, 0) mm, rotated rx -180 ry 0 rz -180 deg; joints [2.634, 0.68, 128.631, -39.311, 90, -87.366]
  Set speed (50.0 mm/s)
  MoveL 169 to (45.6, 20.68, 0) mm, rotated rx -180 ry 0 rz -180 deg; joints [2.291, 0.029, 129.288, -39.316, 90, -87.709]
  MoveL 170 to (44.95, 15.25, 0) mm, rotated rx -180 ry 0 rz 180 deg; joints [1.4, 0.215, 129.101, -39.316, 90, -88.6]
  MoveL 171 to (40.17, 13.45, 0) mm, rotated rx -180 ry 0 rz -180 deg; joints [1.119, -0.521, 129.834, -39.313, 90, -88.881]
  MoveL 172 to (36.57, 10.06, 0) mm, rotated rx -180 ry 0 rz -180 deg; joints [0.563, -0.954, 130.26, -39.305, 90, -89.437]
  MoveL 173 to (35.06, 5.02, 0) mm, rotated rx -180 ry 0 rz -180 deg; joints [-0.281, -0.905, 130.211, -39.307, 90, -90.281]
  MoveL 174 to (29.65, 4.22, 0) mm, rotated rx -180 ry 0 rz -180 deg; joints [-0.422, -1.811, 131.088, -39.277, 90, -90.422]
  MoveL 175 to (27.24, 0, 0) mm, rotated rx -180 ry 0 rz -180 deg; joints [-1.147, -1.957, 131.227, -39.271, 90, -91.147]
  MoveL 176 to (29.65, -4.22, 0) mm, rotated rx -180 ry 0 rz -180 deg; joints [-1.851, -1.238, 130.536, -39.298, 90, -91.851]
  MoveL 177 to (35.06, -5.02, 0) mm, rotated rx -180 ry 0 rz -180 deg; joints [-1.956, -0.242, 129.558, -39.316, 90, -91.956]
  MoveL 178 to (36.57, -10.06, 0) mm, rotated rx -180 ry 0 rz -180 deg; joints [-2.775, 0.361, 128.954, -39.315, 90, -92.775]
  MoveL 179 to (40.17, -13.45, 0) mm, rotated rx -180 ry 0 rz -180 deg; joints [-3.295, 1.201, 128.098, -39.299, 90, -93.295]
  MoveL 180 to (44.95, -15.25, 0) mm, rotated rx -180 ry 0 rz -180 deg; joints [-3.538, 2.12, 127.143, -39.263, 90, -93.538]
  MoveL 181 to (45.6, -20.68, 0) mm, rotated rx -180 ry 0 rz -180 deg; joints [-4.392, 2.601, 126.635, -39.236, 90, -94.392]
  MoveL 182 to (50, -22.96, 0) mm, rotated rx -180 ry 0 rz -180 deg; joints [-4.694, 3.471, 125.702, -39.173, 90, -94.694]
  Set speed (1000.0 mm/s)
  MoveL 183 to (50, -22.96, 0) mm, rotated rx -180 ry 0 rz -180 deg; joints [-4.694, 3.471, 125.702, -39.173, 90, -94.694]
  MoveL 184 to (50, -22.96, 100) mm, rotated rx -180 ry 0 rz -180 deg; joints [-4.694, -6.117, 113.937, -17.82, 90, -94.694]
  Set speed (1000.0 mm/s)
  MoveL 185 to (50, -13.71, 100) mm, rotated rx -180 ry 0 rz 180 deg; joints [-3.247, -6.795, 114.531, -17.736, 90, -93.247]
  MoveL 186 to (50, -13.71, 0) mm, rotated rx -180 ry 0 rz 180 deg; joints [-3.247, 2.849, 126.371, -39.22, 90, -93.247]
  MoveL 187 to (50, -13.71, 0) mm, rotated rx -180 ry 0 rz 180 deg; joints [-3.247, 2.849, 126.371, -39.22, 90, -93.247]
  Set speed (50.0 mm/s)
  MoveL 188 to (46.56, -13.35, 0) mm, rotated rx -180 ry 0 rz -180 deg; joints [-3.22, 2.258, 126.997, -39.256, 90, -93.22]
  MoveL 189 to (45.35, -10.35, 0) mm, rotated rx -180 ry 0 rz 180 deg; joints [-2.754, 1.859, 127.416, -39.275, 90, -92.754]
  MoveL 190 to (45.22, -6.89, 0) mm, rotated rx -180 ry 0 rz 180 deg; joints [-2.2, 1.61, 127.675, -39.285, 90, -92.2]
  MoveL 191 to (43.44, -4.62, 0) mm, rotated rx -180 ry 0 rz 180 deg; joints [-1.844, 1.163, 128.138, -39.3, 90, -91.844]
  MoveL 192 to (39.98, -4.45, 0) mm, rotated rx -180 ry 0 rz -180 deg; joints [-1.834, 0.563, 128.75, -39.313, 90, -91.834]
  MoveL 193 to (36.83, -3.42, 0) mm, rotated rx -180 ry 0 rz -180 deg; joints [-1.681, -0.045, 129.362, -39.316, 90, -91.681]
  MoveL 194 to (36.42, 0, 0) mm, rotated rx -180 ry 0 rz -180 deg; joints [-1.116, -0.342, 129.657, -39.315, 90, -91.116]
  MoveL 195 to (36.83, 3.42, 0) mm, rotated rx -180 ry 0 rz -180 deg; joints [-0.547, -0.492, 129.805, -39.313, 90, -90.547]
  MoveL 196 to (39.98, 4.45, 0) mm, rotated rx -180 ry 0 rz -180 deg; joints [-0.373, -0.008, 129.324, -39.316, 90, -90.373]
  MoveL 197 to (43.44, 4.62, 0) mm, rotated rx -180 ry 0 rz 180 deg; joints [-0.341, 0.58, 128.732, -39.312, 90, -90.341]
  MoveL 198 to (45.22, 6.89, 0) mm, rotated rx -180 ry 0 rz -180 deg; joints [0.031, 0.75, 128.56, -39.31, 90, -89.969]
  MoveL 199 to (45.35, 10.35, 0) mm, rotated rx -180 ry 0 rz -180 deg; joints [0.596, 0.568, 128.745, -39.312, 90, -89.404]
  MoveL 200 to (46.56, 13.35, 0) mm, rotated rx -180 ry 0 rz -180 deg; joints [1.082, 0.604, 128.708, -39.312, 90, -88.918]
  MoveL 201 to (50, 13.71, 0) mm, rotated rx -180 ry 0 rz -180 deg; joints [1.13, 1.179, 128.12, -39.3, 90, -88.87]
  Set speed (1000.0 mm/s)
  MoveL 202 to (50, 13.71, 0) mm, rotated rx -180 ry 0 rz -180 deg; joints [1.13, 1.179, 128.12, -39.3, 90, -88.87]
  MoveL 203 to (50, 13.71, 100) mm, rotated rx -180 ry 0 rz -180 deg; joints [1.13, -8.605, 116.071, -17.467, 90, -88.87]
  Set speed (1000.0 mm/s)
  MoveL 204 to (50, 4.55, 100) mm, rotated rx -180 ry 0 rz -180 deg; joints [-0.346, -8.035, 115.593, -17.558, 90, -90.346]
  MoveL 205 to (50, 4.55, 0) mm, rotated rx -180 ry 0 rz -180 deg; joints [-0.346, 1.706, 127.575, -39.282, 90, -90.346]
  MoveL 206 to (50, 4.55, 0) mm, rotated rx -180 ry 0 rz -180 deg; joints [-0.346, 1.706, 127.575, -39.282, 90, -90.346]
  Set speed (50.0 mm/s)
  MoveL 207 to (47.55, 4.49, 0) mm, rotated rx -180 ry 0 rz -180 deg; joints [-0.357, 1.293, 128.003, -39.296, 90, -90.357]
  MoveL 208 to (46.33, 4.39, 0) mm, rotated rx -180 ry 0 rz -180 deg; joints [-0.375, 1.091, 128.211, -39.302, 90, -90.375]
  MoveL 209 to (45.46, 3.67, 0) mm, rotated rx -180 ry 0 rz -180 deg; joints [-0.493, 0.986, 128.319, -39.305, 90, -90.493]
  MoveL 210 to (45.34, 2.45, 0) mm, rotated rx -180 ry 0 rz -180 deg; joints [-0.691, 1.039, 128.264, -39.303, 90, -90.691]
  MoveL 211 to (45.3, 1.23, 0) mm, rotated rx -180 ry 0 rz -180 deg; joints [-0.89, 1.109, 128.192, -39.302, 90, -90.89]
  MoveL 212 to (45.34, -2.45, 0) mm, rotated rx -180 ry 0 rz -180 deg; joints [-1.484, 1.345, 127.95, -39.295, 90, -91.484]
  MoveL 213 to (45.46, -3.67, 0) mm, rotated rx -180 ry 0 rz -180 deg; joints [-1.68, 1.443, 127.848, -39.291, 90, -91.68]
  MoveL 214 to (46.33, -4.39, 0) mm, rotated rx -180 ry 0 rz -180 deg; joints [-1.792, 1.636, 127.649, -39.284, 90, -91.792]
  MoveL 215 to (47.55, -4.49, 0) mm, rotated rx -180 ry 0 rz -180 deg; joints [-1.802, 1.847, 127.428, -39.276, 90, -91.802]
  MoveL 216 to (48.78, -4.53, 0) mm, rotated rx -180 ry 0 rz 180 deg; joints [-1.802, 2.055, 127.211, -39.266, 90, -91.802]
  MoveL 217 to (50, -4.55, 0) mm, rotated rx -180 ry 0 rz -180 deg; joints [-1.799, 2.261, 126.994, -39.255, 90, -91.799]
  Set speed (1000.0 mm/s)
  MoveL 218 to (50, -4.55, 0) mm, rotated rx -180 ry 0 rz -180 deg; joints [-1.799, 2.261, 126.994, -39.255, 90, -91.799]
  MoveL 219 to (50, -4.55, 100) mm, rotated rx -180 ry 0 rz -180 deg; joints [-1.799, -7.434, 115.082, -17.648, 90, -91.799]
  Set speed (1000.0 mm/s)
  MoveL 220 to (32.32, -50, 100) mm, rotated rx -180 ry 0 rz -180 deg; joints [-9.241, -6.948, 114.664, -17.715, 90, -99.241]
  MoveL 221 to (32.32, -50, 0) mm, rotated rx -180 ry 0 rz -180 deg; joints [-9.241, 2.708, 126.521, -39.229, 90, -99.241]
  MoveL 222 to (32.32, -50, 0) mm, rotated rx -180 ry 0 rz -180 deg; joints [-9.241, 2.708, 126.521, -39.229, 90, -99.241]
  Set speed (50.0 mm/s)
  MoveL 223 to (27.84, -45.4, 0) mm, rotated rx -180 ry 0 rz -180 deg; joints [-8.628, 1.618, 127.667, -39.285, 90, -98.628]
  MoveL 224 to (22.82, -41.5, 0) mm, rotated rx -180 ry 0 rz -180 deg; joints [-8.121, 0.482, 128.831, -39.314, 90, -98.121]
  MoveL 225 to (18.38, -36.52, 0) mm, rotated rx -180 ry 0 rz -180 deg; joints [-7.405, -0.669, 129.98, -39.311, 90, -97.405]
  MoveL 226 to (13.57, -31.87, 0) mm, rotated rx -180 ry 0 rz 180 deg; joints [-6.726, -1.874, 131.149, -39.274, 90, -96.726]
  MoveL 227 to (0, -18.05, 0) mm, rotated rx -180 ry 0 rz -180 deg; joints [-4.549, -5.467, 134.428, -38.961, 90, -94.549]
  MoveL 228 to (-4.47, -22.58, 0) mm, rotated rx -180 ry 0 rz -180 deg; joints [-5.437, -5.88, 134.785, -38.905, 90, -95.437]
  MoveL 229 to (-18.38, -36.52, 0) mm, rotated rx -180 ry 0 rz -180 deg; joints [-8.287, -7.049, 135.775, -38.727, 90, -98.287]
  MoveL 230 to (-22.82, -41.5, 0) mm, rotated rx -180 ry 0 rz -180 deg; joints [-9.328, -7.323, 136.003, -38.68, 90, -99.328]
  MoveL 231 to (-27.84, -45.4, 0) mm, rotated rx -180 ry 0 rz -180 deg; joints [-10.207, -7.796, 136.392, -38.596, 90, -100.207]
  MoveL 232 to (-32.32, -50, 0) mm, rotated rx -180 ry 0 rz -180 deg; joints [-11.215, -8.072, 136.616, -38.544, 90, -101.215]
  Set speed (1000.0 mm/s)
  MoveL 233 to (-32.32, -50, 0) mm, rotated rx -180 ry 0 rz -180 deg; joints [-11.215, -8.072, 136.616, -38.544, 90, -101.215]
  MoveL 234 to (-32.32, -50, 100) mm, rotated rx -180 ry 0 rz -180 deg; joints [-11.215, -18.315, 123.295, -14.979, 90, -101.215]
  Set speed (1000.0 mm/s)
  MoveL 235 to (-22.96, -50, 100) mm, rotated rx -180 ry 0 rz -180 deg; joints [-10.881, -16.624, 122.16, -15.536, 90, -100.881]
  MoveL 236 to (-22.96, -50, 0) mm, rotated rx -180 ry 0 rz -180 deg; joints [-10.881, -6.416, 135.244, -38.827, 90, -100.881]
  MoveL 237 to (-22.96, -50, 0) mm, rotated rx -180 ry 0 rz -180 deg; joints [-10.881, -6.416, 135.244, -38.827, 90, -100.881]
  Set speed (50.0 mm/s)
  MoveL 238 to (-20.68, -45.6, 0) mm, rotated rx -180 ry 0 rz -180 deg; joints [-10.011, -6.496, 135.311, -38.815, 90, -100.011]
  MoveL 239 to (-15.25, -44.95, 0) mm, rotated rx -180 ry 0 rz -180 deg; joints [-9.723, -5.61, 134.552, -38.942, 90, -99.723]
  MoveL 240 to (-13.45, -40.17, 0) mm, rotated rx -180 ry 0 rz -180 deg; joints [-8.814, -5.787, 134.705, -38.918, 90, -98.814]
  MoveL 241 to (-10.06, -36.57, 0) mm, rotated rx -180 ry 0 rz -180 deg; joints [-8.079, -5.55, 134.5, -38.95, 90, -98.079]
  MoveL 242 to (-5.02, -35.06, 0) mm, rotated rx -180 ry 0 rz -180 deg; joints [-7.686, -4.805, 133.847, -39.042, 90, -97.686]
  MoveL 243 to (-4.22, -29.65, 0) mm, rotated rx -180 ry 0 rz 180 deg; joints [-6.705, -5.176, 134.174, -38.998, 90, -96.705]
  MoveL 244 to (0, -27.24, 0) mm, rotated rx -180 ry 0 rz -180 deg; joints [-6.19, -4.646, 133.705, -39.059, 90, -96.19]
  MoveL 245 to (4.22, -29.65, 0) mm, rotated rx -180 ry 0 rz -180 deg; joints [-6.532, -3.682, 132.837, -39.155, 90, -96.532]
  MoveL 246 to (5.02, -35.06, 0) mm, rotated rx -180 ry 0 rz -180 deg; joints [-7.453, -3.055, 132.26, -39.205, 90, -97.453]
  MoveL 247 to (10.06, -36.57, 0) mm, rotated rx -180 ry 0 rz -180 deg; joints [-7.597, -2.06, 131.326, -39.266, 90, -97.597]
  MoveL 248 to (13.45, -40.17, 0) mm, rotated rx -180 ry 0 rz 180 deg; joints [-8.122, -1.175, 130.475, -39.3, 90, -98.122]
  MoveL 249 to (15.25, -44.95, 0) mm, rotated rx -180 ry 0 rz 180 deg; joints [-8.868, -0.456, 129.769, -39.314, 90, -98.868]
  MoveL 250 to (20.68, -45.6, 0) mm, rotated rx -180 ry 0 rz -180 deg; joints [-8.837, 0.486, 128.828, -39.314, 90, -98.837]
  MoveL 251 to (22.96, -50, 0) mm, rotated rx -180 ry 0 rz -180 deg; joints [-9.485, 1.231, 128.067, -39.298, 90, -99.485]
  Set speed (1000.0 mm/s)
  MoveL 252 to (22.96, -50, 0) mm, rotated rx -180 ry 0 rz -180 deg; joints [-9.485, 1.231, 128.067, -39.298, 90, -99.485]
  MoveL 253 to (22.96, -50, 100) mm, rotated rx -180 ry 0 rz -180 deg; joints [-9.485, -8.549, 116.025, -17.476, 90, -99.485]
  Set speed (1000.0 mm/s)
  MoveL 254 to (13.71, -50, 100) mm, rotated rx -180 ry 0 rz 180 deg; joints [-9.738, -10.146, 117.335, -17.188, 90, -99.738]
  MoveL 255 to (13.71, -50, 0) mm, rotated rx -180 ry 0 rz 180 deg; joints [-9.738, -0.254, 129.569, -39.316, 90, -99.738]
  MoveL 256 to (13.71, -50, 0) mm, rotated rx -180 ry 0 rz 180 deg; joints [-9.738, -0.254, 129.569, -39.316, 90, -99.738]
  Set speed (50.0 mm/s)
  MoveL 257 to (13.35, -46.56, 0) mm, rotated rx -180 ry 0 rz -180 deg; joints [-9.184, -0.623, 129.934, -39.312, 90, -99.184]
  MoveL 258 to (10.35, -45.35, 0) mm, rotated rx -180 ry 0 rz -180 deg; joints [-9.063, -1.223, 130.522, -39.298, 90, -99.063]
  MoveL 259 to (6.89, -45.22, 0) mm, rotated rx -180 ry 0 rz -180 deg; joints [-9.134, -1.809, 131.086, -39.277, 90, -99.134]
  MoveL 260 to (4.62, -43.44, 0) mm, rotated rx -180 ry 0 rz -180 deg; joints [-8.894, -2.354, 131.604, -39.25, 90, -98.894]
  MoveL 261 to (4.45, -39.98, 0) mm, rotated rx -180 ry 0 rz -180 deg; joints [-8.309, -2.704, 131.933, -39.229, 90, -98.309]
  MoveL 262 to (3.42, -36.83, 0) mm, rotated rx -180 ry 0 rz -180 deg; joints [-7.794, -3.169, 132.366, -39.197, 90, -97.794]
  MoveL 263 to (0, -36.42, 0) mm, rotated rx -180 ry 0 rz -180 deg; joints [-7.804, -3.798, 132.942, -39.144, 90, -97.804]
  MoveL 264 to (-3.42, -36.83, 0) mm, rotated rx -180 ry 0 rz -180 deg; joints [-7.959, -4.354, 133.445, -39.091, 90, -97.959]
  MoveL 265 to (-4.45, -39.98, 0) mm, rotated rx -180 ry 0 rz -180 deg; joints [-8.537, -4.23, 133.333, -39.103, 90, -98.537]
  MoveL 266 to (-4.62, -43.44, 0) mm, rotated rx -180 ry 0 rz 180 deg; joints [-9.146, -3.922, 133.055, -39.133, 90, -99.146]
  MoveL 267 to (-6.89, -45.22, 0) mm, rotated rx -180 ry 0 rz -180 deg; joints [-9.521, -4.135, 133.248, -39.113, 90, -99.521]
  MoveL 268 to (-10.35, -45.35, 0) mm, rotated rx -180 ry 0 rz -180 deg; joints [-9.647, -4.717, 133.769, -39.051, 90, -99.647]
  MoveL 269 to (-13.35, -46.56, 0) mm, rotated rx -180 ry 0 rz -180 deg; joints [-9.951, -5.111, 134.116, -39.006, 90, -99.951]
  MoveL 270 to (-13.71, -50, 0) mm, rotated rx -180 ry 0 rz 180 deg; joints [-10.569, -4.814, 133.855, -39.04, 90, -100.569]
  Set speed (1000.0 mm/s)
  MoveL 271 to (-13.71, -50, 0) mm, rotated rx -180 ry 0 rz 180 deg; joints [-10.569, -4.814, 133.855, -39.04, 90, -100.569]
  MoveL 272 to (-13.71, -50, 100) mm, rotated rx -180 ry 0 rz 180 deg; joints [-10.569, -14.966, 120.998, -16.032, 90, -100.569]
  Set speed (1000.0 mm/s)
  MoveL 273 to (-4.55, -50, 100) mm, rotated rx -180 ry 0 rz -180 deg; joints [-10.277, -13.341, 119.811, -16.47, 90, -100.277]
  MoveL 274 to (-4.55, -50, 0) mm, rotated rx -180 ry 0 rz -180 deg; joints [-10.277, -3.262, 132.451, -39.19, 90, -100.277]
  MoveL 275 to (-4.55, -50, 0) mm, rotated rx -180 ry 0 rz -180 deg; joints [-10.277, -3.262, 132.451, -39.19, 90, -100.277]
  Set speed (50.0 mm/s)
  MoveL 276 to (-4.49, -47.55, 0) mm, rotated rx -180 ry 0 rz 180 deg; joints [-9.854, -3.495, 132.666, -39.171, 90, -99.854]
  MoveL 277 to (-4.39, -46.33, 0) mm, rotated rx -180 ry 0 rz 180 deg; joints [-9.64, -3.598, 132.76, -39.162, 90, -99.64]
  MoveL 278 to (-3.67, -45.46, 0) mm, rotated rx -180 ry 0 rz -180 deg; joints [-9.469, -3.561, 132.726, -39.165, 90, -99.469]
  MoveL 279 to (-2.45, -45.34, 0) mm, rotated rx -180 ry 0 rz -180 deg; joints [-9.413, -3.366, 132.548, -39.181, 90, -99.413]
  MoveL 280 to (-1.23, -45.3, 0) mm, rotated rx -180 ry 0 rz -180 deg; joints [-9.372, -3.162, 132.359, -39.197, 90, -99.372]
  MoveL 281 to (2.45, -45.34, 0) mm, rotated rx -180 ry 0 rz 180 deg; joints [-9.275, -2.54, 131.779, -39.239, 90, -99.275]
  MoveL 282 to (3.67, -45.46, 0) mm, rotated rx -180 ry 0 rz -180 deg; joints [-9.262, -2.324, 131.576, -39.252, 90, -99.262]
  MoveL 283 to (4.39, -46.33, 0) mm, rotated rx -180 ry 0 rz -180 deg; joints [-9.389, -2.122, 131.384, -39.263, 90, -99.389]
  MoveL 284 to (4.49, -47.55, 0) mm, rotated rx -180 ry 0 rz -180 deg; joints [-9.592, -1.99, 131.259, -39.269, 90, -99.592]
  MoveL 285 to (4.53, -48.78, 0) mm, rotated rx -180 ry 0 rz -180 deg; joints [-9.796, -1.868, 131.143, -39.275, 90, -99.796]
  MoveL 286 to (4.55, -50, 0) mm, rotated rx -180 ry 0 rz -180 deg; joints [-10.001, -1.749, 131.029, -39.28, 90, -100.001]
  Set speed (1000.0 mm/s)
  MoveL 287 to (4.55, -50, 0) mm, rotated rx -180 ry 0 rz -180 deg; joints [-10.001, -1.749, 131.029, -39.28, 90, -100.001]
  MoveL 288 to (4.55, -50, 100) mm, rotated rx -180 ry 0 rz -180 deg; joints [-10.001, -11.741, 118.595, -16.853, 90, -100.001]
  Set speed (1000.0 mm/s)
  MoveL 289 to (4.55, 50, 100) mm, rotated rx -180 ry 0 rz -180 deg; joints [8.156, -19.747, 124.216, -14.469, 90, -81.844]
  MoveL 290 to (4.55, 50, 0) mm, rotated rx -180 ry 0 rz -180 deg; joints [8.156, -9.491, 137.743, -38.252, 90, -81.844]
  MoveL 291 to (4.55, 50, 0) mm, rotated rx -180 ry 0 rz -180 deg; joints [8.156, -9.491, 137.743, -38.252, 90, -81.844]
  Set speed (50.0 mm/s)
  MoveL 292 to (4.49, 47.55, 0) mm, rotated rx -180 ry 0 rz -180 deg; joints [7.689, -9.369, 137.648, -38.279, 90, -82.311]
  MoveL 293 to (4.39, 46.33, 0) mm, rotated rx -180 ry 0 rz -180 deg; joints [7.459, -9.322, 137.611, -38.289, 90, -82.541]
  MoveL 294 to (3.67, 45.46, 0) mm, rotated rx -180 ry 0 rz -180 deg; joints [7.311, -9.426, 137.692, -38.266, 90, -82.689]
  MoveL 295 to (2.45, 45.34, 0) mm, rotated rx -180 ry 0 rz -180 deg; joints [7.317, -9.677, 137.888, -38.21, 90, -82.683]
  MoveL 296 to (1.23, 45.3, 0) mm, rotated rx -180 ry 0 rz -180 deg; joints [7.341, -9.937, 138.088, -38.151, 90, -82.659]
  MoveL 297 to (-2.45, 45.34, 0) mm, rotated rx -180 ry 0 rz -180 deg; joints [7.44, -10.733, 138.692, -37.959, 90, -82.56]
  MoveL 298 to (-3.67, 45.46, 0) mm, rotated rx -180 ry 0 rz -180 deg; joints [7.495, -11.006, 138.896, -37.89, 90, -82.505]
  MoveL 299 to (-4.39, 46.33, 0) mm, rotated rx -180 ry 0 rz -180 deg; joints [7.685, -11.217, 139.052, -37.835, 90, -82.315]
  MoveL 300 to (-4.49, 47.55, 0) mm, rotated rx -180 ry 0 rz -180 deg; joints [7.928, -11.312, 139.122, -37.81, 90, -82.072]
  MoveL 301 to (-4.53, 48.78, 0) mm, rotated rx -180 ry 0 rz 180 deg; joints [8.171, -11.393, 139.182, -37.789, 90, -81.829]
  MoveL 302 to (-4.55, 50, 0) mm, rotated rx -180 ry 0 rz 180 deg; joints [8.414, -11.469, 139.238, -37.769, 90, -81.586]
  Set speed (1000.0 mm/s)
  MoveL 303 to (-4.55, 50, 0) mm, rotated rx -180 ry 0 rz 180 deg; joints [8.414, -11.469, 139.238, -37.769, 90, -81.586]
  MoveL 304 to (-4.55, 50, 100) mm, rotated rx -180 ry 0 rz 180 deg; joints [8.414, -21.713, 125.422, -13.71, 90, -81.586]
  Set speed (1000.0 mm/s)
  MoveL 305 to (-13.71, 50, 100) mm, rotated rx -180 ry 0 rz -180 deg; joints [8.69, -23.734, 126.595, -12.861, 90, -81.31]
  MoveL 306 to (-13.71, 50, 0) mm, rotated rx -180 ry 0 rz -180 deg; joints [8.69, -13.542, 140.713, -37.171, 90, -81.31]
  MoveL 307 to (-13.71, 50, 0) mm, rotated rx -180 ry 0 rz -180 deg; joints [8.69, -13.542, 140.713, -37.171, 90, -81.31]
  Set speed (50.0 mm/s)
  MoveL 308 to (-13.35, 46.56, 0) mm, rotated rx -180 ry 0 rz -180 deg; joints [7.978, -13.241, 140.504, -37.263, 90, -82.022]
  MoveL 309 to (-10.35, 45.35, 0) mm, rotated rx -180 ry 0 rz -180 deg; joints [7.651, -12.484, 139.971, -37.488, 90, -82.349]
  MoveL 310 to (-6.89, 45.22, 0) mm, rotated rx -180 ry 0 rz -180 deg; joints [7.532, -11.701, 139.408, -37.707, 90, -82.468]
  MoveL 311 to (-4.62, 43.44, 0) mm, rotated rx -180 ry 0 rz -180 deg; joints [7.122, -11.09, 138.958, -37.868, 90, -82.878]
  MoveL 312 to (-4.45, 39.98, 0) mm, rotated rx -180 ry 0 rz -180 deg; joints [6.437, -10.835, 138.768, -37.933, 90, -83.563]
  MoveL 313 to (-3.42, 36.83, 0) mm, rotated rx -180 ry 0 rz -180 deg; joints [5.799, -10.41, 138.448, -38.038, 90, -84.201]
  MoveL 314 to (0, 36.42, 0) mm, rotated rx -180 ry 0 rz -180 deg; joints [5.653, -9.655, 137.87, -38.215, 90, -84.347]
  MoveL 315 to (3.42, 36.83, 0) mm, rotated rx -180 ry 0 rz -180 deg; joints [5.667, -8.963, 137.329, -38.366, 90, -84.333]
  MoveL 316 to (4.45, 39.98, 0) mm, rotated rx -180 ry 0 rz -180 deg; joints [6.246, -8.94, 137.311, -38.371, 90, -83.754]
  MoveL 317 to (4.62, 43.44, 0) mm, rotated rx -180 ry 0 rz -180 deg; joints [6.902, -9.108, 137.444, -38.335, 90, -83.098]
  MoveL 318 to (6.89, 45.22, 0) mm, rotated rx -180 ry 0 rz 180 deg; joints [7.187, -8.733, 137.147, -38.414, 90, -82.813]
  MoveL 319 to (10.35, 45.35, 0) mm, rotated rx -180 ry 0 rz -180 deg; joints [7.13, -8.02, 136.575, -38.554, 90, -82.87]
  MoveL 320 to (13.35, 46.56, 0) mm, rotated rx -180 ry 0 rz 180 deg; joints [7.284, -7.47, 136.125, -38.654, 90, -82.716]
  MoveL 321 to (13.71, 50, 0) mm, rotated rx -180 ry 0 rz -180 deg; joints [7.913, -7.574, 136.21, -38.636, 90, -82.087]
  Set speed (1000.0 mm/s)
  MoveL 322 to (13.71, 50, 0) mm, rotated rx -180 ry 0 rz -180 deg; joints [7.913, -7.574, 136.21, -38.636, 90, -82.087]
  MoveL 323 to (13.71, 50, 100) mm, rotated rx -180 ry 0 rz -180 deg; joints [7.913, -17.809, 122.96, -15.151, 90, -82.087]
  Set speed (1000.0 mm/s)
  MoveL 324 to (22.96, 50, 100) mm, rotated rx -180 ry 0 rz -180 deg; joints [7.681, -15.89, 121.652, -15.762, 90, -82.319]
  MoveL 325 to (22.96, 50, 0) mm, rotated rx -180 ry 0 rz -180 deg; joints [7.681, -5.705, 134.634, -38.929, 90, -82.319]
  MoveL 326 to (22.96, 50, 0) mm, rotated rx -180 ry 0 rz -180 deg; joints [7.681, -5.705, 134.634, -38.929, 90, -82.319]
  Set speed (50.0 mm/s)
  MoveL 327 to (20.68, 45.6, 0) mm, rotated rx -180 ry 0 rz -180 deg; joints [6.941, -5.941, 134.838, -38.897, 90, -83.059]
  MoveL 328 to (15.25, 44.95, 0) mm, rotated rx -180 ry 0 rz 180 deg; joints [6.942, -6.998, 135.733, -38.735, 90, -83.058]
  MoveL 329 to (13.45, 40.17, 0) mm, rotated rx -180 ry 0 rz -180 deg; joints [6.099, -7.102, 135.82, -38.718, 90, -83.901]
  MoveL 330 to (10.06, 36.57, 0) mm, rotated rx -180 ry 0 rz -180 deg; joints [5.495, -7.579, 136.215, -38.635, 90, -84.505]
  MoveL 331 to (5.02, 35.06, 0) mm, rotated rx -180 ry 0 rz -180 deg; joints [5.301, -8.52, 136.977, -38.457, 90, -84.699]
  MoveL 332 to (4.22, 29.65, 0) mm, rotated rx -180 ry 0 rz -180 deg; joints [4.29, -8.339, 136.832, -38.493, 90, -85.71]
  MoveL 333 to (0, 27.24, 0) mm, rotated rx -180 ry 0 rz -180 deg; joints [3.888, -9.046, 137.394, -38.349, 90, -86.112]
  MoveL 334 to (-4.22, 29.65, 0) mm, rotated rx -180 ry 0 rz -180 deg; joints [4.414, -10.096, 138.209, -38.113, 90, -85.586]
  MoveL 335 to (-5.02, 35.06, 0) mm, rotated rx -180 ry 0 rz -180 deg; joints [5.484, -10.637, 138.62, -37.983, 90, -84.516]
  MoveL 336 to (-10.06, 36.57, 0) mm, rotated rx -180 ry 0 rz -180 deg; joints [5.882, -11.837, 139.506, -37.67, 90, -84.118]
  MoveL 337 to (-13.45, 40.17, 0) mm, rotated rx -180 ry 0 rz -180 deg; joints [6.681, -12.838, 140.222, -37.384, 90, -83.319]
  MoveL 338 to (-15.25, 44.95, 0) mm, rotated rx -180 ry 0 rz -180 deg; joints [7.702, -13.572, 140.733, -37.161, 90, -82.298]
  MoveL 339 to (-20.68, 45.6, 0) mm, rotated rx -180 ry 0 rz -180 deg; joints [7.993, -14.886, 141.619, -36.734, 90, -82.007]
  MoveL 340 to (-22.96, 50, 0) mm, rotated rx -180 ry 0 rz -180 deg; joints [8.989, -15.731, 142.171, -36.44, 90, -81.011]
  Set speed (1000.0 mm/s)
  MoveL 341 to (-22.96, 50, 0) mm, rotated rx -180 ry 0 rz -180 deg; joints [8.989, -15.731, 142.171, -36.44, 90, -81.011]
  MoveL 342 to (-22.96, 50, 100) mm, rotated rx -180 ry 0 rz -180 deg; joints [8.989, -25.823, 127.736, -11.913, 90, -81.011]
  Set speed (1000.0 mm/s)
  MoveL 343 to (-32.32, 50, 100) mm, rotated rx 180 ry 0 rz -180 deg; joints [9.314, -27.983, 128.841, -10.858, 90, -80.686]
  MoveL 344 to (-32.32, 50, 0) mm, rotated rx -180 ry 0 rz -180 deg; joints [9.314, -18.05, 143.609, -35.559, 90, -80.686]
  MoveL 345 to (-32.32, 50, 0) mm, rotated rx -180 ry 0 rz -180 deg; joints [9.314, -18.05, 143.609, -35.559, 90, -80.686]
  Set speed (50.0 mm/s)
  MoveL 346 to (-27.84, 45.4, 0) mm, rotated rx -180 ry 0 rz -180 deg; joints [8.165, -16.595, 142.719, -36.124, 90, -81.835]
  MoveL 347 to (-22.82, 41.5, 0) mm, rotated rx -180 ry 0 rz -180 deg; joints [7.191, -15.1, 141.761, -36.661, 90, -82.809]
  MoveL 348 to (-18.38, 36.52, 0) mm, rotated rx -180 ry 0 rz -180 deg; joints [6.048, -13.701, 140.822, -37.121, 90, -83.952]
  MoveL 349 to (-13.57, 31.87, 0) mm, rotated rx -180 ry 0 rz -180 deg; joints [5.005, -12.277, 139.824, -37.547, 90, -84.995]
  MoveL 350 to (0, 18.05, 0) mm, rotated rx -180 ry 0 rz -180 deg; joints [2.139, -8.393, 136.876, -38.482, 90, -87.861]
  MoveL 351 to (4.47, 22.58, 0) mm, rotated rx -180 ry 0 rz 180 deg; joints [2.955, -7.812, 136.405, -38.593, 90, -87.045]
  MoveL 352 to (18.38, 36.52, 0) mm, rotated rx -180 ry 0 rz -180 deg; joints [5.341, -5.912, 134.813, -38.901, 90, -84.659]
  MoveL 353 to (22.82, 41.5, 0) mm, rotated rx -180 ry 0 rz -180 deg; joints [6.158, -5.308, 134.29, -38.981, 90, -83.842]
  MoveL 354 to (27.84, 45.4, 0) mm, rotated rx -180 ry 0 rz -180 deg; joints [6.751, -4.527, 133.599, -39.072, 90, -83.249]
  MoveL 355 to (32.32, 50, 0) mm, rotated rx -180 ry 0 rz -180 deg; joints [7.461, -3.878, 133.015, -39.137, 90, -82.539]
  Set speed (1000.0 mm/s)
  MoveL 356 to (32.32, 50, 0) mm, rotated rx -180 ry 0 rz -180 deg; joints [7.461, -3.878, 133.015, -39.137, 90, -82.539]
  MoveL 357 to (32.32, 50, 100) mm, rotated rx -180 ry 0 rz -180 deg; joints [7.461, -13.988, 120.289, -16.301, 90, -82.539]
  Set speed (1000.0 mm/s)
  MoveL 358 to (42.13, 50, 100) mm, rotated rx -180 ry 0 rz -180 deg; joints [7.244, -12.032, 118.819, -16.787, 90, -82.756]
  MoveL 359 to (42.13, 50, 0) mm, rotated rx -180 ry 0 rz -180 deg; joints [7.244, -2.023, 131.29, -39.268, 90, -82.756]
  MoveL 360 to (42.13, 50, 0) mm, rotated rx -180 ry 0 rz -180 deg; joints [7.244, -2.023, 131.29, -39.268, 90, -82.756]
  Set speed (50.0 mm/s)
  MoveL 361 to (35.49, 45.03, 0) mm, rotated rx -180 ry 0 rz -180 deg; joints [6.531, -3.046, 132.252, -39.206, 90, -83.469]
  MoveL 362 to (30.21, 38.5, 0) mm, rotated rx -180 ry 0 rz -180 deg; joints [5.494, -3.729, 132.88, -39.151, 90, -84.506]
  MoveL 363 to (23.42, 33.12, 0) mm, rotated rx -180 ry 0 rz -180 deg; joints [4.651, -4.74, 133.789, -39.049, 90, -85.349]
  MoveL 364 to (17.54, 26.96, 0) mm, rotated rx -180 ry 0 rz 180 deg; joints [3.623, -5.516, 134.47, -38.954, 90, -86.377]
  MoveL 365 to (12.08, 20.31, 0) mm, rotated rx -180 ry 0 rz 180 deg; joints [2.467, -6.153, 135.02, -38.866, 90, -87.533]
  MoveL 366 to (5.14, 15.34, 0) mm, rotated rx -180 ry 0 rz -180 deg; joints [1.599, -7.17, 135.876, -38.706, 90, -88.401]
  MoveL 367 to (0, 8.95, 0) mm, rotated rx -180 ry 0 rz -180 deg; joints [0.421, -7.707, 136.319, -38.612, 90, -89.579]
  MoveL 368 to (-5.14, 15.34, 0) mm, rotated rx -180 ry 0 rz -180 deg; joints [1.654, -9.236, 137.544, -38.308, 90, -88.346]
  MoveL 369 to (-12.08, 20.31, 0) mm, rotated rx -180 ry 0 rz 180 deg; joints [2.673, -11.072, 138.945, -37.873, 90, -87.327]
  MoveL 370 to (-17.54, 26.96, 0) mm, rotated rx -180 ry 0 rz -180 deg; joints [4.074, -12.784, 140.184, -37.4, 90, -85.926]
  MoveL 371 to (-23.42, 33.12, 0) mm, rotated rx -180 ry 0 rz -180 deg; joints [5.447, -14.603, 141.432, -36.829, 90, -84.553]
  MoveL 372 to (-30.21, 38.5, 0) mm, rotated rx -180 ry 0 rz -180 deg; joints [6.745, -16.644, 142.75, -36.106, 90, -83.255]
  MoveL 373 to (-35.49, 45.03, 0) mm, rotated rx -180 ry 0 rz -180 deg; joints [8.327, -18.48, 143.864, -35.384, 90, -81.673]
  MoveL 374 to (-42.13, 50, 0) mm, rotated rx -180 ry 0 rz -180 deg; joints [9.682, -20.609, 145.074, -34.465, 90, -80.318]
  Set speed (1000.0 mm/s)
  MoveL 375 to (-42.13, 50, 0) mm, rotated rx -180 ry 0 rz -180 deg; joints [9.682, -20.609, 145.074, -34.465, 90, -80.318]
  MoveL 376 to (-42.13, 50, 100) mm, rotated rx -180 ry 0 rz -180 deg; joints [9.682, -30.301, 129.946, -9.644, 90, -80.318]

--- Python program Prog3 ---
from robodk.robolink import *  # API to communicate with RoboDK
from robodk.robomath import *  # basic matrix operations

# Any interaction with RoboDK must be done through RDK:
RDK = Robolink()

# Select a robot (popup is displayed if more than one robot is available)
robot = RDK.ItemUserPick('Select a robot', ITEM_TYPE_ROBOT)
if not robot.Valid():
    raise Exception('No robot selected or available')

# get the current position of the TCP with respect to the reference frame:
# (4x4 matrix representing position and orientation)
target_ref = robot.Pose()
pos_ref = target_ref.Pos()
print("Drawing a polygon around the target: ")
print(Pose_2_TxyzRxyz(target_ref))

# move the robot to the first point:
robot.MoveJ(target_ref)

# It is important to provide the reference frame and the tool frames when generating programs offline
robot.setPoseFrame(robot.PoseFrame())
robot.setPoseTool(robot.PoseTool())
robot.setRounding(10)  # Set the rounding parameter (Also known as: CNT, APO/C_DIS, ZoneData, Blending radius, cornering, ...)
robot.setSpeed(200)  # Set linear speed in mm/s

# Set the number of sides of the polygon:
n_sides = 6
R = 100

# make a hexagon around reference target:
for i in range(n_sides + 1):
    ang = i * 2 * pi / n_sides  #angle: 0, 60, 120, ...

    #-----------------------------
    # Movement relative to the reference frame
    # Create a copy of the target
    target_i = Mat(target_ref)
    pos_i = target_i.Pos()
    pos_i[0] = pos_i[0] + R * cos(ang)
    pos_i[1] = pos_i[1] + R * sin(ang)
    target_i.setPos(pos_i)
    print("Moving to target %i: angle %.1f" % (i, ang * 180 / pi))
    print(str(Pose_2_TxyzRxyz(target_i)))
    robot.MoveL(target_i)

    #-----------------------------
    # Post multiply: relative to the tool
    #target_i = target_ref * rotz(ang) * transl(R,0,0) * rotz(-ang)
    #robot.MoveL(target_i)

# move back to the center, then home:
robot.MoveL(target_ref)

print('Done')
